// TIA Portal V19 export
FUNCTION_BLOCK "Axis_EncoderSelection_FB"   // FB29, LAD
TITLE = ENCODER SELECTION PROCEDURE
// stored: Access Published, MemoryReserve 100, SetENOAutomatically false
   VAR_INPUT
      OptionON : Bool := FALSE;
      Execute : Bool := FALSE;
      Rst : Bool := TRUE;
      SelectMotorEncoder : Bool := TRUE;
      Ax_Sts_PM : "TAx_Pos_Sts";
      Ax_Sts_SIEMENS : "TAx_STATUSWORD";
   END_VAR
   VAR_OUTPUT
      Ready : Bool;
      Running : Bool;
      Done : Bool;
      MotorEncoderIsActive : Bool;
      MeasWheelEncoderIsActive : Bool;
      AlarmsPresence : Bool;
      WarningPresence : Bool;
      Ctrl_ForceAxPowerOff : Bool;
   END_VAR
   VAR_IN_OUT
      TO_Ax : TO_PositioningAxis;
      Persistent_EncoderSelection_OK : Bool;
   END_VAR
   VAR
      Status : Int;
      Alarm : Struct
         TOut_AxisPowerRemoving : Bool;
         TOut_WaitCndEncoderChange : Bool;
         TOut_WaitDoneEncoderChange : Bool;
         Error_MC_SetSensor : Bool;
         ErrorId_MC_SetSensor : Word;
         Error_NoEncoderChange : Bool;
      END_STRUCT;
      Warning : Struct
         EncInUseNeedToBeChanged : Bool;
      END_STRUCT;
      TON_TimeOutInit : TON_TIME;
      My_SetSensor : MC_SETSENSOR;
   END_VAR
   VAR CONSTANT
      MOTOR_ENCODER_NUMBER : Int := 1;
      MWHEEL_ENCODER_NUMBER : Int := 2;
   END_VAR
BEGIN

REGION Network 1: Status Active Encoder
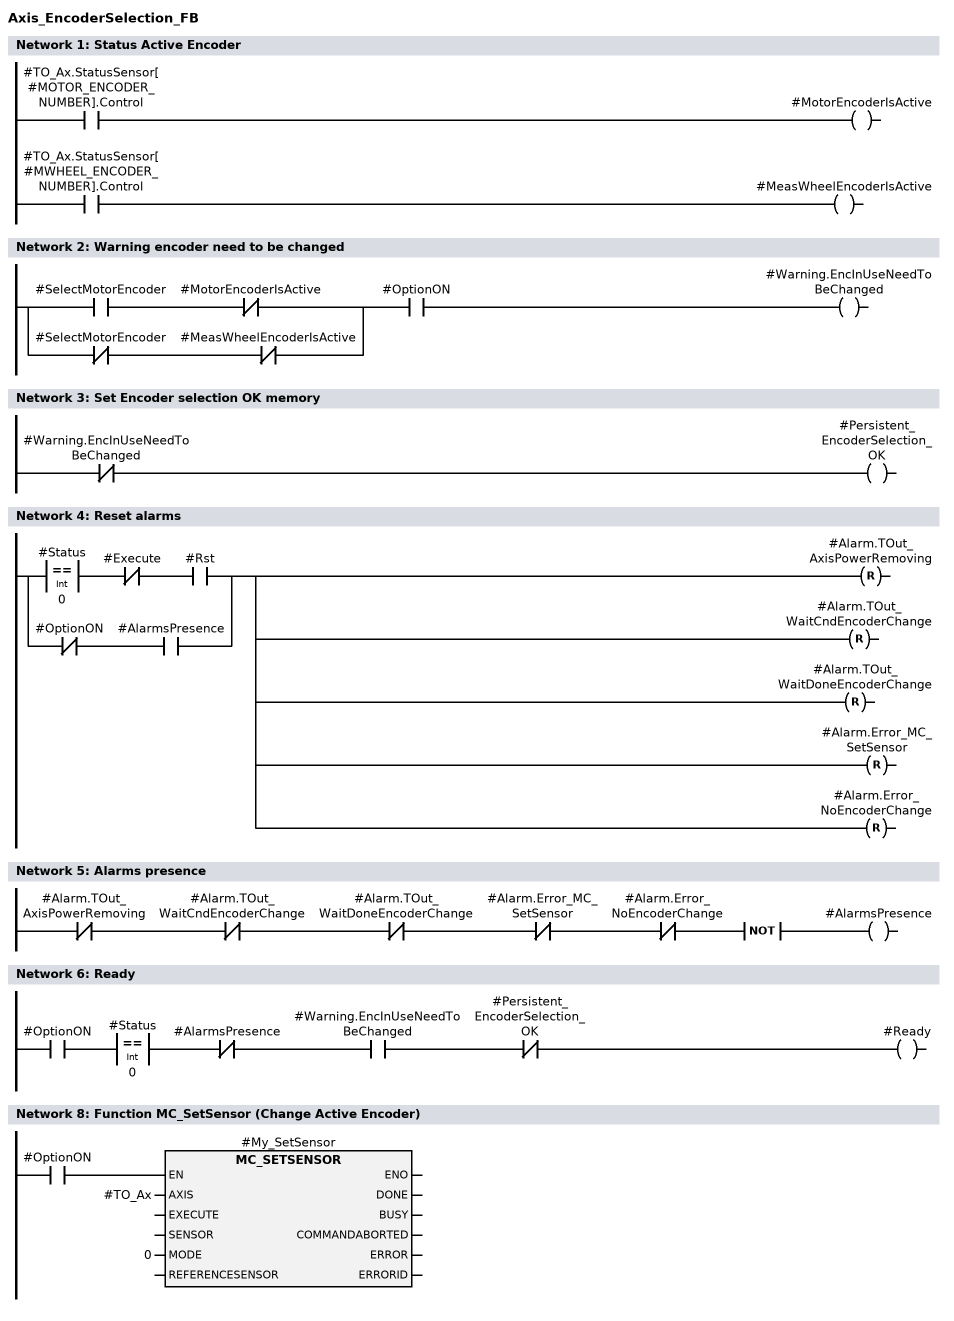
   RUNG wire#powerrail
      Contact( #TO_Ax.StatusSensor[#MOTOR_ENCODER_NUMBER].Control )
      Coil( #MotorEncoderIsActive )
   END_RUNG
   RUNG wire#powerrail
      Contact( #TO_Ax.StatusSensor[#MWHEEL_ENCODER_NUMBER].Control )
      Coil( #MeasWheelEncoderIsActive )
   END_RUNG
   // the same network as SCL:
   #MotorEncoderIsActive := #TO_Ax.StatusSensor[#MOTOR_ENCODER_NUMBER].Control;
   #MeasWheelEncoderIsActive := #TO_Ax.StatusSensor[#MWHEEL_ENCODER_NUMBER].Control;
END_REGION

REGION Network 2: Warning encoder need to be changed
   RUNG wire#powerrail
      Contact( #SelectMotorEncoder )
      I_Contact( #MotorEncoderIsActive )
      wire#w1
      Contact( #OptionON )
      Coil( #Warning.EncInUseNeedToBeChanged )
   END_RUNG
   RUNG wire#powerrail
      I_Contact( #SelectMotorEncoder )
      I_Contact( #MeasWheelEncoderIsActive )
   END_RUNG wire#w1
   // the same network as SCL:
   #Warning.EncInUseNeedToBeChanged := ((#SelectMotorEncoder AND NOT #MotorEncoderIsActive) OR (NOT #SelectMotorEncoder AND NOT #MeasWheelEncoderIsActive)) AND #OptionON;
END_REGION

REGION Network 3: Set Encoder selection OK memory
   RUNG wire#powerrail
      I_Contact( #Warning.EncInUseNeedToBeChanged )
      Coil( #Persistent_EncoderSelection_OK )
   END_RUNG
   // the same network as SCL:
   #Persistent_EncoderSelection_OK := NOT #Warning.EncInUseNeedToBeChanged;
END_REGION

REGION Network 4: Reset alarms
   RUNG wire#powerrail
      { S7_Templates := "SrcType := Int" } EQ_Contact(in1 := #Status, in2 := 0)
      I_Contact( #Execute )
      Contact( #Rst )
      wire#w1
      R_Coil( #Alarm.TOut_AxisPowerRemoving )
   END_RUNG
   RUNG wire#powerrail
      I_Contact( #OptionON )
      Contact( #AlarmsPresence )
   END_RUNG wire#w1
   RUNG wire#w1
      R_Coil( #Alarm.TOut_WaitCndEncoderChange )
   END_RUNG
   RUNG wire#w1
      R_Coil( #Alarm.TOut_WaitDoneEncoderChange )
   END_RUNG
   RUNG wire#w1
      R_Coil( #Alarm.Error_MC_SetSensor )
   END_RUNG
   RUNG wire#w1
      R_Coil( #Alarm.Error_NoEncoderChange )
   END_RUNG
   // the same network as SCL:
   IF ((#Status = 0) AND NOT #Execute AND #Rst) OR (NOT #OptionON AND #AlarmsPresence) THEN
       #Alarm.TOut_AxisPowerRemoving := FALSE;
       #Alarm.TOut_WaitCndEncoderChange := FALSE;
       #Alarm.TOut_WaitDoneEncoderChange := FALSE;
       #Alarm.Error_MC_SetSensor := FALSE;
       #Alarm.Error_NoEncoderChange := FALSE;
   END_IF;
END_REGION

REGION Network 5: Alarms presence
   RUNG wire#powerrail
      I_Contact( #Alarm.TOut_AxisPowerRemoving )
      I_Contact( #Alarm.TOut_WaitCndEncoderChange )
      I_Contact( #Alarm.TOut_WaitDoneEncoderChange )
      I_Contact( #Alarm.Error_MC_SetSensor )
      I_Contact( #Alarm.Error_NoEncoderChange )
      Not()
      Coil( #AlarmsPresence )
   END_RUNG
   // the same network as SCL:
   #AlarmsPresence := NOT (NOT #Alarm.TOut_AxisPowerRemoving AND NOT #Alarm.TOut_WaitCndEncoderChange AND NOT #Alarm.TOut_WaitDoneEncoderChange AND NOT #Alarm.Error_MC_SetSensor AND NOT #Alarm.Error_NoEncoderChange);
END_REGION

REGION Network 6: Ready
   RUNG wire#powerrail
      Contact( #OptionON )
      { S7_Templates := "SrcType := Int" } EQ_Contact(in1 := #Status, in2 := 0)
      I_Contact( #AlarmsPresence )
      Contact( #Warning.EncInUseNeedToBeChanged )
      I_Contact( #Persistent_EncoderSelection_OK )
      Coil( #Ready )
   END_RUNG
   // the same network as SCL:
   #Ready := #OptionON AND (#Status = 0) AND NOT #AlarmsPresence AND #Warning.EncInUseNeedToBeChanged AND NOT #Persistent_EncoderSelection_OK;
END_REGION

REGION Network 7 (SCL): Sequence
   CASE #Status OF

       //=============================================================================================
       // STATUS = 0 IDLE
       //=============================================================================================
       //
       0:

           #TON_TimeOutInit(IN:=FALSE,PT:=T#1s);


           #Ctrl_ForceAxPowerOff := FALSE;

           #My_SetSensor.Execute := FALSE;

           #Running := FALSE;
           #Done := FALSE;


           IF  #Ready AND #Execute THEN

               #Running := TRUE;
               #Ready := FALSE;


               #Status += 1;

           END_IF;




       //=============================================================================================
       //  STATUS 1 - STOP AXIS REMOVING POWER
       //=============================================================================================
       //
       1:

           #TON_TimeOutInit(IN:=TRUE,PT:=T#10s);

           #Ctrl_ForceAxPowerOff := TRUE;


           IF  #TON_TimeOutInit.Q THEN

               #Alarm.TOut_AxisPowerRemoving := TRUE;
               #Status := 0;


           ELSIF   NOT #Ax_Sts_PM.Enabled AND #Ax_Sts_PM.Standstill THEN

               #TON_TimeOutInit(IN:=FALSE,PT:=T#10s);

               #Status += 1;
           END_IF;




       //=============================================================================================
       // STATUS 2 - START SELECTION DESIRED ENCODER
       //=============================================================================================
       //
       2:

           #TON_TimeOutInit(IN:=TRUE,PT:=T#1s);

           IF    #TON_TimeOutInit.Q THEN

               #Alarm.TOut_WaitCndEncoderChange := TRUE;

               #Status := 0;


           ELSIF   NOT #My_SetSensor.Done
               AND
               NOT #My_SetSensor.Busy
               AND
               NOT #My_SetSensor.Error
               AND
               NOT #My_SetSensor.Execute THEN

               #My_SetSensor.Execute := TRUE;


               IF  #SelectMotorEncoder THEN
                   #My_SetSensor.Sensor := #MOTOR_ENCODER_NUMBER;
               ELSE
                   #My_SetSensor.Sensor := #MWHEEL_ENCODER_NUMBER;
               END_IF;

               #Status += 1;
           END_IF;



       //=============================================================================================
       // STATUS 3 - CHECK EXECUTION OF MC_SETSENSOR
       //=============================================================================================
       //
       3:

           #TON_TimeOutInit(IN:=TRUE,PT:=T#1s);

           IF    #TON_TimeOutInit.Q THEN

               #Alarm.TOut_WaitDoneEncoderChange := TRUE;

               #Status := 0;

           ELSIF      #My_SetSensor.Error THEN

               #Alarm.Error_MC_SetSensor := TRUE;
               #Alarm.ErrorId_MC_SetSensor := #My_SetSensor.ErrorId;
               #Status := 0;


           ELSIF #My_SetSensor.Done THEN

               #TON_TimeOutInit(IN:=FALSE,PT:=T#1s);

               #My_SetSensor.Execute := false;
               #Status += 1;


           END_IF;


       //=============================================================================================
       // STATUS 4 - CHECK CHANGE OF SELECTED ENCODER
       //=============================================================================================
       //
       4:

           IF  #Warning.EncInUseNeedToBeChanged THEN

               #Alarm.Error_NoEncoderChange := TRUE;
               #Status := 0;
           ELSE
               #Status += 1;
           END_IF;



       //=============================================================================================
       // STATUS 5 - DONE
       //=============================================================================================
       //   
       5:

           #Ctrl_ForceAxPowerOff := FALSE;
           #My_SetSensor.Execute := FALSE;


           #Done := TRUE;

           IF NOT #Execute THEN
               #Status := 0;
           END_IF;


       ELSE
           #Status := 0;

   END_CASE;
END_REGION

REGION Network 8: Function MC_SetSensor (Change Active Encoder)
   RUNG wire#powerrail
      Contact( #OptionON )
      #My_SetSensor.MC_SETSENSOR(Axis := #TO_Ax, Execute :=, Sensor :=, Mode := 0, ReferenceSensor :=, Done =>, Busy =>, CommandAborted =>, Error =>, ErrorId =>)
   END_RUNG
   // the same network as SCL:
   IF #OptionON THEN
       #My_SetSensor(Axis := #TO_Ax, Mode := 0);   // MC_SETSENSOR
   END_IF;
END_REGION

REGION Network 9: >
END_REGION

REGION Network 10: >
END_REGION
END_FUNCTION_BLOCK
